{attribute 'pack_mode' := '2'}
TYPE U_XTS_TRANSPORT_CTRL :
UNION
  stCtrl              : ST_XTS_TRANSPORT_CTRL;
  byCtrl    AT %Q*    : ARRAY[1..SIZEOF(ST_XTS_TRANSPORT_CTRL)] OF BYTE;
END_UNION
END_TYPE

(* stored: Version 1.1.0.1
   DUT U_XTS_TRANSPORT_CTRL: Id {e2d8980f-cf1e-4aae-a226-4cdc2a65f9e1} *)
